Omron CX-Programmer project NewProject (CX-Programmer 9.61)

# PLC NewPLC1: CP1E N30

## Global symbols (name address type ; comment)
0.00 BOOL  ; PB1
0.01 BOOL  ; PB1
0.02 BOOL  ; PB2
100.00 BOOL  ; LAMP
100.01 BOOL  ; LAMP2

## Program NewProgram1 (cyclic task 0)

### Section Section1

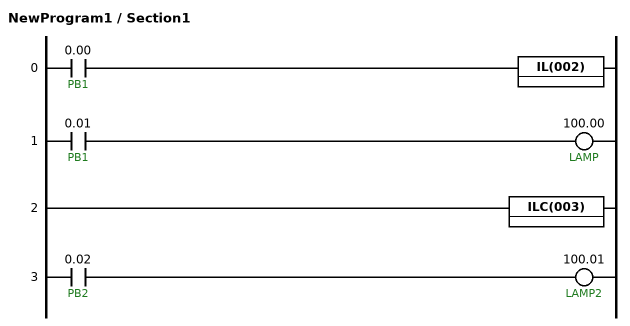
; rung 0
LD 0.00  ; PB1
IL(002)
; rung 1
LD 0.01  ; PB1
OUT 100.00  ; LAMP
; rung 2
ILC(003)
; rung 3
LD 0.02  ; PB2
OUT 100.01  ; LAMP2

### Section END
; rung 0
END(001)